// TIA Portal V19 export
DATA_BLOCK "AccRollConveyor_PERS"   // DB153
// stored: MemoryReserve 100
   VAR RETAIN
      PersistentValues : "udt_AccRollConveyor_Pers";
   END_VAR
BEGIN
   PersistentValues.Data.MaterialPresence_S2_Entry := FALSE;
   PersistentValues.Data.MaterialPresence_S3 := TRUE;
   PersistentValues.Data.MaterialPresence_S4 := FALSE;
   PersistentValues.Data.MaterialPresence_S5_Stop := FALSE;
   PersistentValues.Data.MaterialPresence_ExitLeft1 := FALSE;
   PersistentValues.Data.MaterialPresence_ExitLeft2 := FALSE;
   PersistentValues.Data.MaterialPresence_ExitLeft3 := FALSE;
   PersistentValues.Data.MaterialPresence_ExitLeft4 := FALSE;
   PersistentValues.Par.UnloadAllLeft := TRUE;
   PersistentValues.Par.S2_DistanceFromstop := 5590.0;
   PersistentValues.Par.S3_DistanceFromstop := 3200.0;
   PersistentValues.Par.S4_DistanceFromstop := 450.0;
   PersistentValues.Par.Rollway_Lenght := 7335.0;
   PersistentValues.Par.Rollway_AutMinSpeed := 10000.0;
   PersistentValues.Par.Rollway_AutAcc := 1000.0;
   PersistentValues.Par.Rollway_AutDec := 1000.0;
   PersistentValues.Par.Rollway_DelayStopRollformer := T#200MS;
   PersistentValues.Par.Rollway_DelaySlowDownRollformer := T#250MS;
   PersistentValues.Par.Rollway_DistanceBetweenPieces := 600.0;
   PersistentValues.Par.Rollway_StopSlowDownSpeed := 2000.0;
   PersistentValues.Par.Pusher_MaxLenghtUseFirst := 5501.0;
   PersistentValues.Par.Pusher_DeltaLenghtForUse := 0.0;
   PersistentValues.Par.Pusher_DistanceFromStop[1] := 228.0;
   PersistentValues.Par.Pusher_DistanceFromStop[2] := 788.0;
   PersistentValues.Par.Pusher_DistanceFromStop[3] := 1348.0;
   PersistentValues.Par.Pusher_DistanceFromStop[4] := 2098.0;
   PersistentValues.Par.Pusher_DistanceFromStop[5] := 3098.0;
   PersistentValues.Par.Pusher_DistanceFromStop[6] := 4478.0;
   PersistentValues.Par.Roll1.Man.VelBwd := 5000.0;
   PersistentValues.Par.Roll1.Man.VelFwdHigh := 5000.0;
   PersistentValues.Par.Roll1.Man.VelFwdLow := 5000.0;
   PersistentValues.Par.Roll1.Man.Acc := 1000.0;
   PersistentValues.Par.Roll1.Man.Dec := 1000.0;
   PersistentValues.Par.Roll1.Man.DelayChangeVel := T#0MS;
   PersistentValues.Par.Roll2.Man.VelBwd := 5000.0;
   PersistentValues.Par.Roll2.Man.VelFwdHigh := 5000.0;
   PersistentValues.Par.Roll2.Man.VelFwdLow := 5000.0;
   PersistentValues.Par.Roll2.Man.Acc := 1000.0;
   PersistentValues.Par.Roll2.Man.Dec := 1000.0;
   PersistentValues.Par.Roll2.Man.DelayChangeVel := T#0MS;
   PersistentValues.Par.Roll3.Man.VelBwd := 5000.0;
   PersistentValues.Par.Roll3.Man.VelFwdHigh := 5000.0;
   PersistentValues.Par.Roll3.Man.VelFwdLow := 5000.0;
   PersistentValues.Par.Roll3.Man.Acc := 1000.0;
   PersistentValues.Par.Roll3.Man.Dec := 1000.0;
   PersistentValues.Par.Roll3.Man.DelayChangeVel := T#0MS;
END_DATA_BLOCK
